FUNCTION_BLOCK GF_Entleeren	EXTENDS FB_Basisfunktionalitaeten
VAR_INPUT
	// Instanzieren von Sensoren mit Interfaces
	Level		:I_Sensor;
	// Instanzieren von Aktoren mit Interfaces
	Ventil		:I_Magnetventil;
	
	// Frage:
	// Wie wird aumgesetzt, dass der Inhalt in ein bestimmten Reaktor läuft
END_VAR
VAR_OUTPUT
	
END_VAR
VAR
	
END_VAR

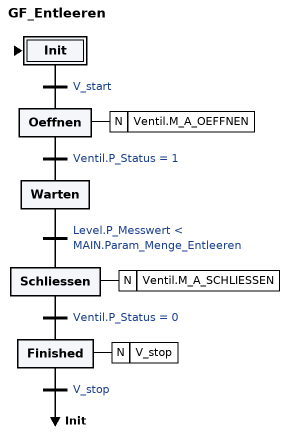
INITIAL_STEP Init:
END_STEP
TRANSITION FROM Init TO Oeffnen
    := V_start;
END_TRANSITION
STEP Oeffnen:
    Ventil.M_A_OEFFNEN(N);
END_STEP
TRANSITION FROM Oeffnen TO Warten
    := Ventil.P_Status = 1;
END_TRANSITION
STEP Warten:
END_STEP
TRANSITION FROM Warten TO Schliessen
    := Level.P_Messwert < MAIN.Param_Menge_Entleeren;
END_TRANSITION
STEP Schliessen:
    Ventil.M_A_SCHLIESSEN(N);
END_STEP
TRANSITION FROM Schliessen TO Finished
    := Ventil.P_Status = 0;
END_TRANSITION
STEP Finished:
    V_stop(N);
END_STEP
TRANSITION FROM Finished TO Init
    := V_stop;
END_TRANSITION

END_FUNCTION_BLOCK

(* stored: Version 1.1.0.1, ProductVersion 3.1.4024.12
   POU GF_Entleeren: Id {c2b92295-fb26-4f0a-8170-9b037e32b2ff}, SpecialFunc None *)
